PROGRAM MAIN
VAR
	tcpclient : TcpClient; 
END_VAR

tcpclient();

END_PROGRAM

(* stored: Version 1.1.0.1, ProductVersion 3.1.4018.2
   POU MAIN: Id {814d40bc-e99d-43b5-b54e-410f57618c41}, SpecialFunc None *)
